{attribute 'enable_dynamic_creation'}
FUNCTION_BLOCK FB_Yellow IMPLEMENTS I_Color
VAR_INPUT
END_VAR
VAR_OUTPUT
END_VAR
VAR
END_VAR


METHOD M_Fill : BOOL
ADSLOGSTR(ADSLOG_MSGTYPE_HINT, 'Paint Yellow', '');
M_Fill := TRUE;
END_METHOD

END_FUNCTION_BLOCK

(* stored: Version 1.1.0.1, ProductVersion 3.1.4024.12
   POU FB_Yellow: Id {0f08c85f-8c65-4f2b-8312-1a34a6ee00f4}, SpecialFunc None
   Method M_Fill: Id {6ad1cfcd-39e4-49fd-b1dc-eea5f3951bdf} *)
